// TIA Portal V17 export
// export: Created 2025-06-26T06:49:08.0055945Z, ExportSetting WithDefaults, DisplayName Totally Integrated Automation Portal, DisplayVersion V17 Update 8, DisplayName TIA Portal Openness, DisplayVersion V17 Update 8, DisplayName TIA Portal Version Control Interface, DisplayVersion V17, DisplayName STEP 7 Professional, DisplayVersion V17 Update 8, DisplayName STEP 7 Safety, DisplayVersion V17 Update 6, DisplayName WinCC Advanced, DisplayVersion V17 Update 8
FUNCTION_BLOCK "Puma"   // FB2, LAD
TITLE = Combine signals from Puma into DB_Application
{ S7_Optimized_Access := 'TRUE' }
VERSION : 0.1
// stored: AutoNumber true, IsIECCheckEnabled false, IsRetainMemResEnabled false, MemoryReserve 100, SetENOAutomatically false, UDAEnableTagReadback false
   VAR_INPUT
      bEnable : Bool;
   END_VAR
   VAR
      Watchdog : "fbHeartbeatCount2";
      Dummy { S7_SetPoint := 'True'} : UInt;
      epForceExpansionValveSP : Bool;
      enForceExpansionValveSP : Bool;
      epForceHeatSinkOutSP : Bool;
      enForceHeatSinkOutSP : Bool;
      epForceMotorRpmSP : Bool;
      enForceMotorRpmSP : Bool;
      epForceOilHeatingSP : Bool;
      enForceOilHeatingSP : Bool;
      epForcePinchSP : Bool;
      enForcePinchSP : Bool;
      epForceSuperheatSP : Bool;
      enForceSuperheatSP : Bool;
      epStartRequest : Bool;
      enStartRequest : Bool;
      epStopRequest : Bool;
      enStopRequest : Bool;
      epAlarmAcknowledge : Bool;
      enAlarmAcknowledge : Bool;
      epResetEmergencyStop : Bool;
      enResetEmergencyStop : Bool;
      epHydrolockProtection : Bool;
      enHydrolockProtection : Bool;
      enClearance : Bool;
      ExpansionManualPrev : Real;
      HeatSinkManualPrev : Real;
      PerformanceManualPrev : Real;
      OilHeatingManualPrev : Real;
      PinchManualPrev : Real;
      SuperheatManualPrev : Real;
      WatchdogTimeout : TON_TIME;
   END_VAR
   VAR_TEMP
      bStopReq : Bool;
      bWatchdogOk : Bool;
   END_VAR
   VAR_TEMP   // added for the SCL form of the ladder/FBD networks
      _w1 : Bool;
      _w2 : Bool;
      _w3 : Bool;
      _w4 : Bool;
      _w5 : Bool;
      _w6 : Bool;
      _w7 : Bool;
      _w8 : Bool;
      _w9 : Bool;
      _w10 : Bool;
      _w11 : Bool;
      _w12 : Bool;
   END_VAR
BEGIN

REGION Network 1: Watchdog
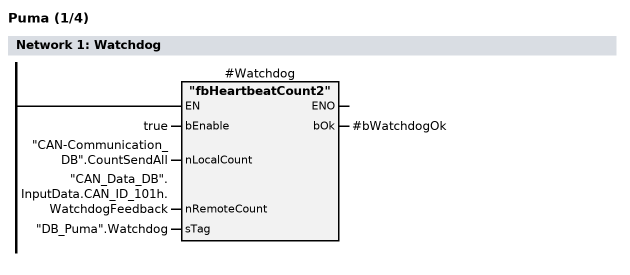
   RUNG wire#powerrail
      #Watchdog(bEnable := true, nLocalCount := "CAN-Communication_DB".CountSendAll, nRemoteCount := "CAN_Data_DB".InputData.CAN_ID_101h.WatchdogFeedback, sTag := "DB_Puma".Watchdog, bOk => #bWatchdogOk)
   END_RUNG
   // the same network as SCL:
   #Watchdog(bEnable := true,   // "fbHeartbeatCount2"
             nLocalCount := "CAN-Communication_DB".CountSendAll,
             nRemoteCount := "CAN_Data_DB".InputData.CAN_ID_101h.WatchdogFeedback,
             sTag := "DB_Puma".Watchdog,
             bOk => #bWatchdogOk);
END_REGION

REGION Network 2: Write Puma setpoints to Application
   // A positive edge followed by a SET  writes to the destination bit once, without "holding" the value. Easiest to write & read in ladder.
   // Triggering a MOVE on value change writes the value once without continually overwriting it.
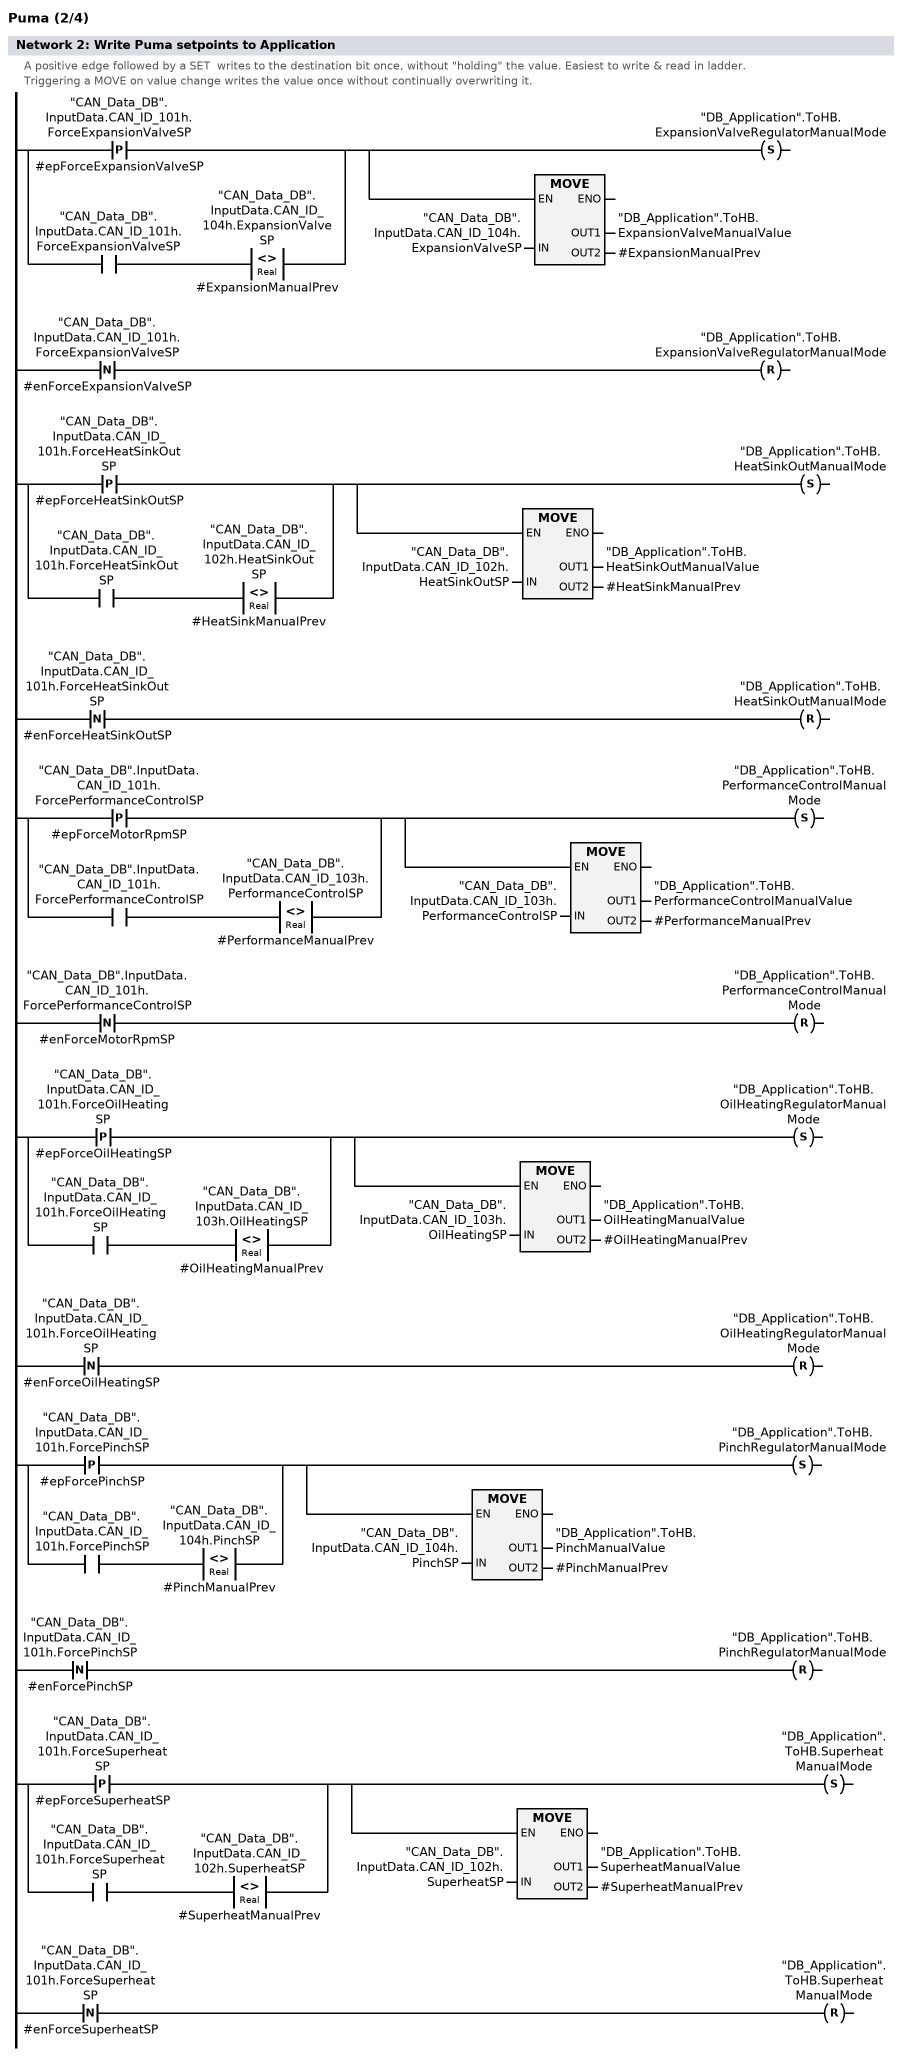
   RUNG wire#powerrail
      P_Contact(operand := "CAN_Data_DB".InputData.CAN_ID_101h.ForceExpansionValveSP, bit := #epForceExpansionValveSP)
      wire#w1
      S_Coil( "DB_Application".ToHB.ExpansionValveRegulatorManualMode )
   END_RUNG
   RUNG wire#powerrail
      Contact( "CAN_Data_DB".InputData.CAN_ID_101h.ForceExpansionValveSP )
      { S7_Templates := "SrcType := Real" } NE_Contact(in1 := "CAN_Data_DB".InputData.CAN_ID_104h.ExpansionValveSP, in2 := #ExpansionManualPrev)
   END_RUNG wire#w1
   RUNG wire#w1
      Move(in := "CAN_Data_DB".InputData.CAN_ID_104h.ExpansionValveSP, out1 => "DB_Application".ToHB.ExpansionValveManualValue, out2 => #ExpansionManualPrev)
   END_RUNG
   RUNG wire#powerrail
      N_Contact(operand := "CAN_Data_DB".InputData.CAN_ID_101h.ForceExpansionValveSP, bit := #enForceExpansionValveSP)
      R_Coil( "DB_Application".ToHB.ExpansionValveRegulatorManualMode )
   END_RUNG
   RUNG wire#powerrail
      P_Contact(operand := "CAN_Data_DB".InputData.CAN_ID_101h.ForceHeatSinkOutSP, bit := #epForceHeatSinkOutSP)
      wire#w2
      S_Coil( "DB_Application".ToHB.HeatSinkOutManualMode )
   END_RUNG
   RUNG wire#powerrail
      Contact( "CAN_Data_DB".InputData.CAN_ID_101h.ForceHeatSinkOutSP )
      { S7_Templates := "SrcType := Real" } NE_Contact(in1 := "CAN_Data_DB".InputData.CAN_ID_102h.HeatSinkOutSP, in2 := #HeatSinkManualPrev)
   END_RUNG wire#w2
   RUNG wire#w2
      Move(in := "CAN_Data_DB".InputData.CAN_ID_102h.HeatSinkOutSP, out1 => "DB_Application".ToHB.HeatSinkOutManualValue, out2 => #HeatSinkManualPrev)
   END_RUNG
   RUNG wire#powerrail
      N_Contact(operand := "CAN_Data_DB".InputData.CAN_ID_101h.ForceHeatSinkOutSP, bit := #enForceHeatSinkOutSP)
      R_Coil( "DB_Application".ToHB.HeatSinkOutManualMode )
   END_RUNG
   RUNG wire#powerrail
      P_Contact(operand := "CAN_Data_DB".InputData.CAN_ID_101h.ForcePerformanceControlSP, bit := #epForceMotorRpmSP)
      wire#w3
      S_Coil( "DB_Application".ToHB.PerformanceControlManualMode )
   END_RUNG
   RUNG wire#powerrail
      Contact( "CAN_Data_DB".InputData.CAN_ID_101h.ForcePerformanceControlSP )
      { S7_Templates := "SrcType := Real" } NE_Contact(in1 := "CAN_Data_DB".InputData.CAN_ID_103h.PerformanceControlSP, in2 := #PerformanceManualPrev)
   END_RUNG wire#w3
   RUNG wire#w3
      Move(in := "CAN_Data_DB".InputData.CAN_ID_103h.PerformanceControlSP, out1 => "DB_Application".ToHB.PerformanceControlManualValue, out2 => #PerformanceManualPrev)
   END_RUNG
   RUNG wire#powerrail
      N_Contact(operand := "CAN_Data_DB".InputData.CAN_ID_101h.ForcePerformanceControlSP, bit := #enForceMotorRpmSP)
      R_Coil( "DB_Application".ToHB.PerformanceControlManualMode )
   END_RUNG
   RUNG wire#powerrail
      P_Contact(operand := "CAN_Data_DB".InputData.CAN_ID_101h.ForceOilHeatingSP, bit := #epForceOilHeatingSP)
      wire#w4
      S_Coil( "DB_Application".ToHB.OilHeatingRegulatorManualMode )
   END_RUNG
   RUNG wire#powerrail
      Contact( "CAN_Data_DB".InputData.CAN_ID_101h.ForceOilHeatingSP )
      { S7_Templates := "SrcType := Real" } NE_Contact(in1 := "CAN_Data_DB".InputData.CAN_ID_103h.OilHeatingSP, in2 := #OilHeatingManualPrev)
   END_RUNG wire#w4
   RUNG wire#w4
      Move(in := "CAN_Data_DB".InputData.CAN_ID_103h.OilHeatingSP, out1 => "DB_Application".ToHB.OilHeatingManualValue, out2 => #OilHeatingManualPrev)
   END_RUNG
   RUNG wire#powerrail
      N_Contact(operand := "CAN_Data_DB".InputData.CAN_ID_101h.ForceOilHeatingSP, bit := #enForceOilHeatingSP)
      R_Coil( "DB_Application".ToHB.OilHeatingRegulatorManualMode )
   END_RUNG
   RUNG wire#powerrail
      P_Contact(operand := "CAN_Data_DB".InputData.CAN_ID_101h.ForcePinchSP, bit := #epForcePinchSP)
      wire#w5
      S_Coil( "DB_Application".ToHB.PinchRegulatorManualMode )
   END_RUNG
   RUNG wire#powerrail
      Contact( "CAN_Data_DB".InputData.CAN_ID_101h.ForcePinchSP )
      { S7_Templates := "SrcType := Real" } NE_Contact(in1 := "CAN_Data_DB".InputData.CAN_ID_104h.PinchSP, in2 := #PinchManualPrev)
   END_RUNG wire#w5
   RUNG wire#w5
      Move(in := "CAN_Data_DB".InputData.CAN_ID_104h.PinchSP, out1 => "DB_Application".ToHB.PinchManualValue, out2 => #PinchManualPrev)
   END_RUNG
   RUNG wire#powerrail
      N_Contact(operand := "CAN_Data_DB".InputData.CAN_ID_101h.ForcePinchSP, bit := #enForcePinchSP)
      R_Coil( "DB_Application".ToHB.PinchRegulatorManualMode )
   END_RUNG
   RUNG wire#powerrail
      P_Contact(operand := "CAN_Data_DB".InputData.CAN_ID_101h.ForceSuperheatSP, bit := #epForceSuperheatSP)
      wire#w6
      S_Coil( "DB_Application".ToHB.SuperheatManualMode )
   END_RUNG
   RUNG wire#powerrail
      Contact( "CAN_Data_DB".InputData.CAN_ID_101h.ForceSuperheatSP )
      { S7_Templates := "SrcType := Real" } NE_Contact(in1 := "CAN_Data_DB".InputData.CAN_ID_102h.SuperheatSP, in2 := #SuperheatManualPrev)
   END_RUNG wire#w6
   RUNG wire#w6
      Move(in := "CAN_Data_DB".InputData.CAN_ID_102h.SuperheatSP, out1 => "DB_Application".ToHB.SuperheatManualValue, out2 => #SuperheatManualPrev)
   END_RUNG
   RUNG wire#powerrail
      N_Contact(operand := "CAN_Data_DB".InputData.CAN_ID_101h.ForceSuperheatSP, bit := #enForceSuperheatSP)
      R_Coil( "DB_Application".ToHB.SuperheatManualMode )
   END_RUNG
   // the same network as SCL:
   #_w1 := "CAN_Data_DB".InputData.CAN_ID_101h.ForceExpansionValveSP AND NOT #epForceExpansionValveSP;   // rising edge of "CAN_Data_DB".InputData.CAN_ID_101h.ForceExpansionValveSP
   #epForceExpansionValveSP := "CAN_Data_DB".InputData.CAN_ID_101h.ForceExpansionValveSP;
   IF #_w1 OR ("CAN_Data_DB".InputData.CAN_ID_101h.ForceExpansionValveSP AND ("CAN_Data_DB".InputData.CAN_ID_104h.ExpansionValveSP <> #ExpansionManualPrev)) THEN
       "DB_Application".ToHB.ExpansionValveRegulatorManualMode := TRUE;
       "DB_Application".ToHB.ExpansionValveManualValue := "CAN_Data_DB".InputData.CAN_ID_104h.ExpansionValveSP;
       #ExpansionManualPrev := "CAN_Data_DB".InputData.CAN_ID_104h.ExpansionValveSP;
   END_IF;
   #_w2 := NOT "CAN_Data_DB".InputData.CAN_ID_101h.ForceExpansionValveSP AND #enForceExpansionValveSP;   // falling edge of "CAN_Data_DB".InputData.CAN_ID_101h.ForceExpansionValveSP
   #enForceExpansionValveSP := "CAN_Data_DB".InputData.CAN_ID_101h.ForceExpansionValveSP;
   IF #_w2 THEN "DB_Application".ToHB.ExpansionValveRegulatorManualMode := FALSE; END_IF;
   #_w3 := "CAN_Data_DB".InputData.CAN_ID_101h.ForceHeatSinkOutSP AND NOT #epForceHeatSinkOutSP;   // rising edge of "CAN_Data_DB".InputData.CAN_ID_101h.ForceHeatSinkOutSP
   #epForceHeatSinkOutSP := "CAN_Data_DB".InputData.CAN_ID_101h.ForceHeatSinkOutSP;
   IF #_w3 OR ("CAN_Data_DB".InputData.CAN_ID_101h.ForceHeatSinkOutSP AND ("CAN_Data_DB".InputData.CAN_ID_102h.HeatSinkOutSP <> #HeatSinkManualPrev)) THEN
       "DB_Application".ToHB.HeatSinkOutManualMode := TRUE;
       "DB_Application".ToHB.HeatSinkOutManualValue := "CAN_Data_DB".InputData.CAN_ID_102h.HeatSinkOutSP;
       #HeatSinkManualPrev := "CAN_Data_DB".InputData.CAN_ID_102h.HeatSinkOutSP;
   END_IF;
   #_w4 := NOT "CAN_Data_DB".InputData.CAN_ID_101h.ForceHeatSinkOutSP AND #enForceHeatSinkOutSP;   // falling edge of "CAN_Data_DB".InputData.CAN_ID_101h.ForceHeatSinkOutSP
   #enForceHeatSinkOutSP := "CAN_Data_DB".InputData.CAN_ID_101h.ForceHeatSinkOutSP;
   IF #_w4 THEN "DB_Application".ToHB.HeatSinkOutManualMode := FALSE; END_IF;
   #_w5 := "CAN_Data_DB".InputData.CAN_ID_101h.ForcePerformanceControlSP AND NOT #epForceMotorRpmSP;   // rising edge of "CAN_Data_DB".InputData.CAN_ID_101h.ForcePerformanceControlSP
   #epForceMotorRpmSP := "CAN_Data_DB".InputData.CAN_ID_101h.ForcePerformanceControlSP;
   IF #_w5 OR ("CAN_Data_DB".InputData.CAN_ID_101h.ForcePerformanceControlSP AND ("CAN_Data_DB".InputData.CAN_ID_103h.PerformanceControlSP <> #PerformanceManualPrev)) THEN
       "DB_Application".ToHB.PerformanceControlManualMode := TRUE;
       "DB_Application".ToHB.PerformanceControlManualValue := "CAN_Data_DB".InputData.CAN_ID_103h.PerformanceControlSP;
       #PerformanceManualPrev := "CAN_Data_DB".InputData.CAN_ID_103h.PerformanceControlSP;
   END_IF;
   #_w6 := NOT "CAN_Data_DB".InputData.CAN_ID_101h.ForcePerformanceControlSP AND #enForceMotorRpmSP;   // falling edge of "CAN_Data_DB".InputData.CAN_ID_101h.ForcePerformanceControlSP
   #enForceMotorRpmSP := "CAN_Data_DB".InputData.CAN_ID_101h.ForcePerformanceControlSP;
   IF #_w6 THEN "DB_Application".ToHB.PerformanceControlManualMode := FALSE; END_IF;
   #_w7 := "CAN_Data_DB".InputData.CAN_ID_101h.ForceOilHeatingSP AND NOT #epForceOilHeatingSP;   // rising edge of "CAN_Data_DB".InputData.CAN_ID_101h.ForceOilHeatingSP
   #epForceOilHeatingSP := "CAN_Data_DB".InputData.CAN_ID_101h.ForceOilHeatingSP;
   IF #_w7 OR ("CAN_Data_DB".InputData.CAN_ID_101h.ForceOilHeatingSP AND ("CAN_Data_DB".InputData.CAN_ID_103h.OilHeatingSP <> #OilHeatingManualPrev)) THEN
       "DB_Application".ToHB.OilHeatingRegulatorManualMode := TRUE;
       "DB_Application".ToHB.OilHeatingManualValue := "CAN_Data_DB".InputData.CAN_ID_103h.OilHeatingSP;
       #OilHeatingManualPrev := "CAN_Data_DB".InputData.CAN_ID_103h.OilHeatingSP;
   END_IF;
   #_w8 := NOT "CAN_Data_DB".InputData.CAN_ID_101h.ForceOilHeatingSP AND #enForceOilHeatingSP;   // falling edge of "CAN_Data_DB".InputData.CAN_ID_101h.ForceOilHeatingSP
   #enForceOilHeatingSP := "CAN_Data_DB".InputData.CAN_ID_101h.ForceOilHeatingSP;
   IF #_w8 THEN "DB_Application".ToHB.OilHeatingRegulatorManualMode := FALSE; END_IF;
   #_w9 := "CAN_Data_DB".InputData.CAN_ID_101h.ForcePinchSP AND NOT #epForcePinchSP;   // rising edge of "CAN_Data_DB".InputData.CAN_ID_101h.ForcePinchSP
   #epForcePinchSP := "CAN_Data_DB".InputData.CAN_ID_101h.ForcePinchSP;
   IF #_w9 OR ("CAN_Data_DB".InputData.CAN_ID_101h.ForcePinchSP AND ("CAN_Data_DB".InputData.CAN_ID_104h.PinchSP <> #PinchManualPrev)) THEN
       "DB_Application".ToHB.PinchRegulatorManualMode := TRUE;
       "DB_Application".ToHB.PinchManualValue := "CAN_Data_DB".InputData.CAN_ID_104h.PinchSP;
       #PinchManualPrev := "CAN_Data_DB".InputData.CAN_ID_104h.PinchSP;
   END_IF;
   #_w10 := NOT "CAN_Data_DB".InputData.CAN_ID_101h.ForcePinchSP AND #enForcePinchSP;   // falling edge of "CAN_Data_DB".InputData.CAN_ID_101h.ForcePinchSP
   #enForcePinchSP := "CAN_Data_DB".InputData.CAN_ID_101h.ForcePinchSP;
   IF #_w10 THEN "DB_Application".ToHB.PinchRegulatorManualMode := FALSE; END_IF;
   #_w11 := "CAN_Data_DB".InputData.CAN_ID_101h.ForceSuperheatSP AND NOT #epForceSuperheatSP;   // rising edge of "CAN_Data_DB".InputData.CAN_ID_101h.ForceSuperheatSP
   #epForceSuperheatSP := "CAN_Data_DB".InputData.CAN_ID_101h.ForceSuperheatSP;
   IF #_w11 OR ("CAN_Data_DB".InputData.CAN_ID_101h.ForceSuperheatSP AND ("CAN_Data_DB".InputData.CAN_ID_102h.SuperheatSP <> #SuperheatManualPrev)) THEN
       "DB_Application".ToHB.SuperheatManualMode := TRUE;
       "DB_Application".ToHB.SuperheatManualValue := "CAN_Data_DB".InputData.CAN_ID_102h.SuperheatSP;
       #SuperheatManualPrev := "CAN_Data_DB".InputData.CAN_ID_102h.SuperheatSP;
   END_IF;
   #_w12 := NOT "CAN_Data_DB".InputData.CAN_ID_101h.ForceSuperheatSP AND #enForceSuperheatSP;   // falling edge of "CAN_Data_DB".InputData.CAN_ID_101h.ForceSuperheatSP
   #enForceSuperheatSP := "CAN_Data_DB".InputData.CAN_ID_101h.ForceSuperheatSP;
   IF #_w12 THEN "DB_Application".ToHB.SuperheatManualMode := FALSE; END_IF;
END_REGION

REGION Network 3: Start request
   // PumaSystemReady: Puma is ok
   // Clearance: Puma and the Test Support System are ok.
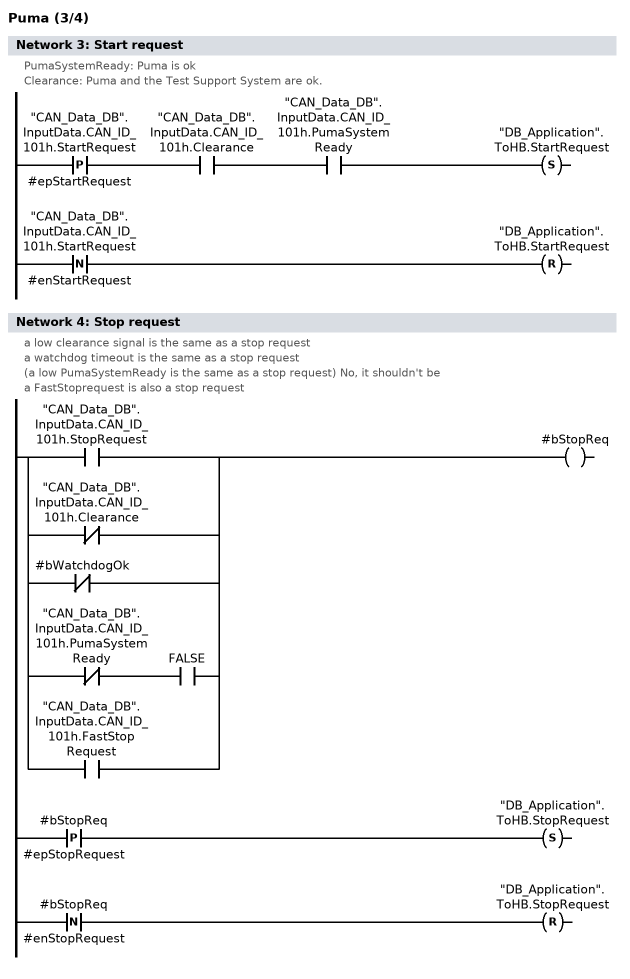
   RUNG wire#powerrail
      P_Contact(operand := "CAN_Data_DB".InputData.CAN_ID_101h.StartRequest, bit := #epStartRequest)
      Contact( "CAN_Data_DB".InputData.CAN_ID_101h.Clearance )
      Contact( "CAN_Data_DB".InputData.CAN_ID_101h.PumaSystemReady )
      S_Coil( "DB_Application".ToHB.StartRequest )
   END_RUNG
   RUNG wire#powerrail
      N_Contact(operand := "CAN_Data_DB".InputData.CAN_ID_101h.StartRequest, bit := #enStartRequest)
      R_Coil( "DB_Application".ToHB.StartRequest )
   END_RUNG
   // the same network as SCL:
   #_w1 := "CAN_Data_DB".InputData.CAN_ID_101h.StartRequest AND NOT #epStartRequest;   // rising edge of "CAN_Data_DB".InputData.CAN_ID_101h.StartRequest
   #epStartRequest := "CAN_Data_DB".InputData.CAN_ID_101h.StartRequest;
   IF #_w1 AND "CAN_Data_DB".InputData.CAN_ID_101h.Clearance AND "CAN_Data_DB".InputData.CAN_ID_101h.PumaSystemReady THEN
       "DB_Application".ToHB.StartRequest := TRUE;
   END_IF;
   #_w2 := NOT "CAN_Data_DB".InputData.CAN_ID_101h.StartRequest AND #enStartRequest;   // falling edge of "CAN_Data_DB".InputData.CAN_ID_101h.StartRequest
   #enStartRequest := "CAN_Data_DB".InputData.CAN_ID_101h.StartRequest;
   IF #_w2 THEN "DB_Application".ToHB.StartRequest := FALSE; END_IF;
END_REGION

REGION Network 4: Stop request
   // a low clearance signal is the same as a stop request
   // a watchdog timeout is the same as a stop request
   // (a low PumaSystemReady is the same as a stop request) No, it shouldn't be
   // a FastStoprequest is also a stop request
   RUNG wire#powerrail
      Contact( "CAN_Data_DB".InputData.CAN_ID_101h.StopRequest )
      wire#w1
      Coil( #bStopReq )
   END_RUNG
   RUNG wire#powerrail
      I_Contact( "CAN_Data_DB".InputData.CAN_ID_101h.Clearance )
   END_RUNG wire#w1
   RUNG wire#powerrail
      I_Contact( #bWatchdogOk )
   END_RUNG wire#w1
   RUNG wire#powerrail
      I_Contact( "CAN_Data_DB".InputData.CAN_ID_101h.PumaSystemReady )
      Contact( FALSE )
   END_RUNG wire#w1
   RUNG wire#powerrail
      Contact( "CAN_Data_DB".InputData.CAN_ID_101h.FastStopRequest )
   END_RUNG wire#w1
   RUNG wire#powerrail
      P_Contact(operand := #bStopReq, bit := #epStopRequest)
      S_Coil( "DB_Application".ToHB.StopRequest )
   END_RUNG
   RUNG wire#powerrail
      N_Contact(operand := #bStopReq, bit := #enStopRequest)
      R_Coil( "DB_Application".ToHB.StopRequest )
   END_RUNG
   // the same network as SCL:
   #bStopReq := "CAN_Data_DB".InputData.CAN_ID_101h.StopRequest OR NOT "CAN_Data_DB".InputData.CAN_ID_101h.Clearance OR NOT #bWatchdogOk OR (NOT "CAN_Data_DB".InputData.CAN_ID_101h.PumaSystemReady AND FALSE) OR "CAN_Data_DB".InputData.CAN_ID_101h.FastStopRequest;
   #_w1 := #bStopReq AND NOT #epStopRequest;   // rising edge of #bStopReq
   #epStopRequest := #bStopReq;
   IF #_w1 THEN "DB_Application".ToHB.StopRequest := TRUE; END_IF;
   #_w2 := NOT #bStopReq AND #enStopRequest;   // falling edge of #bStopReq
   #enStopRequest := #bStopReq;
   IF #_w2 THEN "DB_Application".ToHB.StopRequest := FALSE; END_IF;
END_REGION

REGION Network 5: Commands
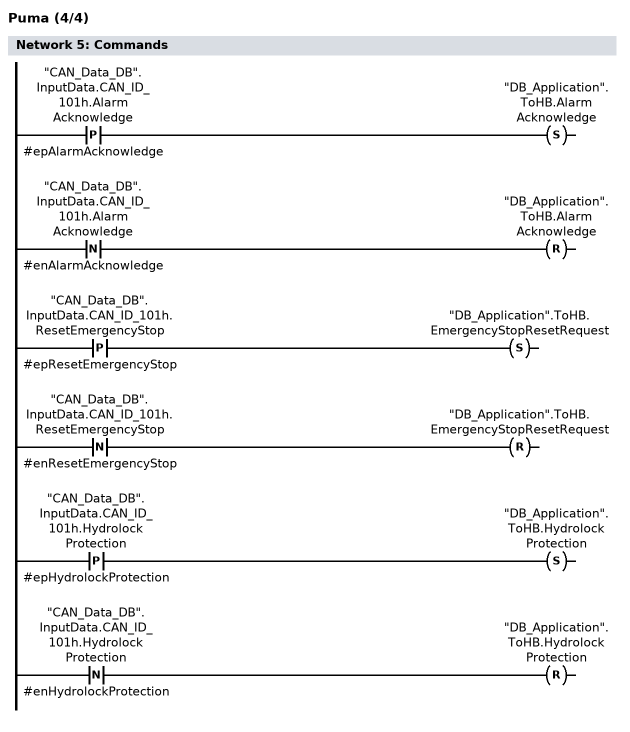
   RUNG wire#powerrail
      P_Contact(operand := "CAN_Data_DB".InputData.CAN_ID_101h.AlarmAcknowledge, bit := #epAlarmAcknowledge)
      S_Coil( "DB_Application".ToHB.AlarmAcknowledge )
   END_RUNG
   RUNG wire#powerrail
      N_Contact(operand := "CAN_Data_DB".InputData.CAN_ID_101h.AlarmAcknowledge, bit := #enAlarmAcknowledge)
      R_Coil( "DB_Application".ToHB.AlarmAcknowledge )
   END_RUNG
   RUNG wire#powerrail
      P_Contact(operand := "CAN_Data_DB".InputData.CAN_ID_101h.ResetEmergencyStop, bit := #epResetEmergencyStop)
      S_Coil( "DB_Application".ToHB.EmergencyStopResetRequest )
   END_RUNG
   RUNG wire#powerrail
      N_Contact(operand := "CAN_Data_DB".InputData.CAN_ID_101h.ResetEmergencyStop, bit := #enResetEmergencyStop)
      R_Coil( "DB_Application".ToHB.EmergencyStopResetRequest )
   END_RUNG
   RUNG wire#powerrail
      P_Contact(operand := "CAN_Data_DB".InputData.CAN_ID_101h.HydrolockProtection, bit := #epHydrolockProtection)
      S_Coil( "DB_Application".ToHB.HydrolockProtection )
   END_RUNG
   RUNG wire#powerrail
      N_Contact(operand := "CAN_Data_DB".InputData.CAN_ID_101h.HydrolockProtection, bit := #enHydrolockProtection)
      R_Coil( "DB_Application".ToHB.HydrolockProtection )
   END_RUNG
   // the same network as SCL:
   #_w1 := "CAN_Data_DB".InputData.CAN_ID_101h.AlarmAcknowledge AND NOT #epAlarmAcknowledge;   // rising edge of "CAN_Data_DB".InputData.CAN_ID_101h.AlarmAcknowledge
   #epAlarmAcknowledge := "CAN_Data_DB".InputData.CAN_ID_101h.AlarmAcknowledge;
   IF #_w1 THEN "DB_Application".ToHB.AlarmAcknowledge := TRUE; END_IF;
   #_w2 := NOT "CAN_Data_DB".InputData.CAN_ID_101h.AlarmAcknowledge AND #enAlarmAcknowledge;   // falling edge of "CAN_Data_DB".InputData.CAN_ID_101h.AlarmAcknowledge
   #enAlarmAcknowledge := "CAN_Data_DB".InputData.CAN_ID_101h.AlarmAcknowledge;
   IF #_w2 THEN "DB_Application".ToHB.AlarmAcknowledge := FALSE; END_IF;
   #_w3 := "CAN_Data_DB".InputData.CAN_ID_101h.ResetEmergencyStop AND NOT #epResetEmergencyStop;   // rising edge of "CAN_Data_DB".InputData.CAN_ID_101h.ResetEmergencyStop
   #epResetEmergencyStop := "CAN_Data_DB".InputData.CAN_ID_101h.ResetEmergencyStop;
   IF #_w3 THEN "DB_Application".ToHB.EmergencyStopResetRequest := TRUE; END_IF;
   #_w4 := NOT "CAN_Data_DB".InputData.CAN_ID_101h.ResetEmergencyStop AND #enResetEmergencyStop;   // falling edge of "CAN_Data_DB".InputData.CAN_ID_101h.ResetEmergencyStop
   #enResetEmergencyStop := "CAN_Data_DB".InputData.CAN_ID_101h.ResetEmergencyStop;
   IF #_w4 THEN "DB_Application".ToHB.EmergencyStopResetRequest := FALSE; END_IF;
   #_w5 := "CAN_Data_DB".InputData.CAN_ID_101h.HydrolockProtection AND NOT #epHydrolockProtection;   // rising edge of "CAN_Data_DB".InputData.CAN_ID_101h.HydrolockProtection
   #epHydrolockProtection := "CAN_Data_DB".InputData.CAN_ID_101h.HydrolockProtection;
   IF #_w5 THEN "DB_Application".ToHB.HydrolockProtection := TRUE; END_IF;
   #_w6 := NOT "CAN_Data_DB".InputData.CAN_ID_101h.HydrolockProtection AND #enHydrolockProtection;   // falling edge of "CAN_Data_DB".InputData.CAN_ID_101h.HydrolockProtection
   #enHydrolockProtection := "CAN_Data_DB".InputData.CAN_ID_101h.HydrolockProtection;
   IF #_w6 THEN "DB_Application".ToHB.HydrolockProtection := FALSE; END_IF;
END_REGION
END_FUNCTION_BLOCK
